TYPE PrintConfig_typ :
STRUCT
	StationEnable	: ARRAY[0..GVL.MULTISTN_NUM_STN - 1] OF BOOL;
	ProcessIndex	: ARRAY[0..GVL.MULTISTN_NUM_STN - 1] OF USINT;
	FinalPrint		: ARRAY[0..GVL.MULTISTN_NUM_STN - 1] OF BOOL;
	LastProcessIndex0StnIndex	: USINT;
END_STRUCT
END_TYPE

(* stored: Version 1.1.0.1, ProductVersion 3.1.4024.12
   DUT PrintConfig_typ: Id {9209a69b-e1e1-0d1c-260d-3f71121896c7} *)
